PROGRAM MAIN
VAR
	{attribute 'OPC.UA.DA' := '1'}
	{attribute 'OPC.UA.DA.StructuredType' := '1'}
	//Simulate virtual axes
	simulated		:	ARRAY [1..GVL.axisNumMax] OF ST_SimulateStage;
	bSimulate		:	ARRAY [1..GVL.axisNumMax] OF BOOL;	//Do we want to simulate?
	
	//{attribute 'OPC.UA.DA' := '0'}
	drives			:	ARRAY [1..GVL.axisNumMax] OF FB_AxisDrive;	
	
	bDisableMC		:	BOOL; 		//boolean control if true the motion control application specific code is disabled - dumb box
	iState			:	UINT;		//state machine index

	(*
		Outputs that are set in the hmi and wired to power axis limit switches. Currently not configred as part of the programme
		Will be added to ST_AxisControl in future
	*)
	limitEnable1	AT %Q*	: BOOL;
	limitEnable2	AT %Q*	: BOOL;	
	
	i: UINT;		//General indexing value for FOR loops	
	
	//HMI VARIABLES	
	hmiAxisSelect	:	UINT:=1;

END_VAR

AXES();
PROG();
//SIMULATE();

ACTION AXES:
FOR GVL.iAxis:=1 TO GVL.axisNumMax DO
	drives[GVL.iAxis](AxisController:=GVL.axes[GVL.iAxis]);
END_FOR
END_ACTION

(*
	Scans through axes (from low to high) checking "done" status
*)
METHOD CheckCoupled : BOOL
VAR_INPUT
	iLow	:	UINT;		//lowest index to check
	iHigh	:	UINT;		//highest index to check
END_VAR

VAR
	i		:	UINT;
END_VAR
CheckCoupled:=TRUE;
FOR i:=iLow TO iHigh BY 1 DO
	CheckCoupled:= CheckCoupled AND (GVL.axes[i].iAxisState=500);
END_FOR
END_METHOD

(*
	Scans through axes (from low to high) checking "done" status
*)
METHOD CheckDone : BOOL
VAR_INPUT
	iLow	:	UINT;		//lowest index to check
	iHigh	:	UINT;		//highest index to check
END_VAR

VAR
	i		:	UINT;
END_VAR
CheckDone:=TRUE;
FOR i:=iLow TO iHigh BY 1 DO
	CheckDone:= CheckDone AND GVL.axes[i].bDone;
END_FOR
END_METHOD

(*
	Scans through axes (from low to high) checking "done" status
*)
METHOD CheckMoving : BOOL
VAR_INPUT
	iLow	:	UINT;		//lowest index to check
	iHigh	:	UINT;		//highest index to check
END_VAR

VAR
	i		:	UINT;
	statiks: INT;
END_VAR
CheckMoving:=FALSE;
FOR i:=iLow TO iHigh BY 1 DO
	CheckMoving:= CheckMoving OR (GVL.axes[i].Axis.status.Moving);
END_FOR
END_METHOD

(*
	Gear out an axis
*)
METHOD GearOut : BOOL
VAR_INPUT
	i	:	UINT;	//Axis index to gear out
END_VAR
GVL.axes[i].eCommand:=eMcCommand.GearOut;
GVL.axes[i].bExecute:=TRUE;
END_METHOD

(*
	Power up a single axis of index i
*)
METHOD PowerUp : BOOL
VAR_INPUT
	i	:	UINT;
END_VAR
GVL.axes[i].bEnable:=TRUE;
GVL.axes[i].fOverride:=100;
Limits.FwLimit[i]:=TRUE;	//Set high as I have no hardware linked
Limits.BwLimit[i]:=TRUE;	//Set high as I have no hardware linked
END_METHOD

ACTION PROG:
CASE iState OF
	0:	//CHECK AXIS ID's are correct. Gearing limits currently requires the assigned array index of an axis to match the NC ID.
		//May be possible to negate this by changing axes to GVLs so that they can be seen within the drives function - CASE 0 NO LONGER REQ
		iState:=1;
		FOR i:=1 TO GVL.axisNumMax BY 1 DO
			IF GVL.axes[i].Axis.NcToPlc.AxisId <> i THEN
				iState:=999;
			END_IF
		END_FOR
		
	1:	//Gear out all axes to begin
		FOR i:=1 TO 8 BY 1 DO
			GearOut(i:=i);
		END_FOR
		iState:= 2;
	2:	//Wait for gear out
		IF CheckDone(iLow:=1, iHigh:=8) THEN
			iState:=3;
		END_IF
	3:	//Power up axes (and set limits true as no hardware connected)
		limitEnable1 	:=	TRUE;
		limitEnable2	:=	TRUE;
		FOR i:=1 TO 8 BY 1 DO
			PowerUp(i:=i);
		END_FOR
		iState:= 4;
		
	4:	//HOMING ROUTING
		
		iState:=	10;
		
		
	10:	//Start of main state loop. Are the blades coupled in to the virtual axes?
		//SlitPositions(North:=1,South:=2,East:=3,West:=4,VG:=5,VC:=6,HG:=7,HC:=8);
		IF NOT CheckCoupled(iLow:=1, iHigh:=4) THEN
			iState:=11;
		END_IF
		
	11:	//Blades are not coupled. Update the virtual positions
		FOR i:=1 TO 8 BY 1 DO
			GearOut(i:=i);
		END_FOR
	
		iState:=12;
			
		
	12:	//Confirm positions set
		IF CheckDone(iLow:=5,iHigh:=8) THEN
			iState:=12;
		END_IF	
		iState:=13;
	
	13:	//Check Moving
		SlitPositions(North:=1,South:=2,East:=3,West:=4,VG:=5,VC:=6,HG:=7,HC:=8);
		iState:=14;
		

	14: //Blades not moving, time to setup again
		IF CheckDone(iLow:=5,iHigh:=8) THEN
			iState:=15;
		END_IF			

		
	15:	//Check movin
		IF CheckMoving(iLow:=1, iHigh:=4) THEN
			iState:= 13;
		ELSE
			iState:=16;
		END_IF
	

	16:	//Multimaster gearin
		SlitSetup(North:=1,South:=2,East:=3,West:=4,VG:=5,VC:=6,HG:=7,HC:=8);
		iState:=17;	
		
	17:
		IF CheckDone(iLow:=1,iHigh:=8) THEN
			iState:=10;
		END_IF
		
	50:
		
	51:
						
			
	100:	//DO NOTHING

		
	
	999: //ERROR
		//INOP STATE	
END_CASE
END_ACTION

ACTION SIMULATE:
(*
Simulate axes if bool set TRUE
*)
FOR i:=1 TO GVL.axisNumMax BY 1 DO
	IF bSimulate[i] THEN
		simulateStage(position:=GVL.axes[i].Axis.NcToPlc.ActPos, iAxis:=i, simulated:=simulated[i]);
		GVL.axes[i].MCSignalRef.Level:=simulated[i].absSw;
	END_IF
END_FOR
END_ACTION

(*
	Basic virtual axis simulation.
	Will trigger limit switches beyond set points
	Will trigger absolute switch between given set points
*)
METHOD simulateStage : BOOL
VAR_INPUT
	position	:	LREAL;		//Axis current position
	iAxis		:	UINT;		//Axis index
END_VAR
VAR_IN_OUT
	simulated	:	ST_SimulateStage;	//Struct to hold simulation parameters
END_VAR
Limits.FwLimit[iAxis]:= position < simulated.fHighLim;
Limits.BwLimit[iAxis]:= position > simulated.fLowLim;

simulated.absSw:= (position < simulated.fHighAbs) AND (position > simulated.fLowAbs);
END_METHOD

(*
	Calculate gap positions of a slit set given N/S/E/W blades
*)
METHOD SlitPositions : BOOL
VAR_INPUT
	North	:	UINT;	//North blade index
	South	:	UINT;	//South blade index
	East	:	UINT;	//East blade index
	West	:	UINT;	//West blade index
	VG		:	UINT;	//Vertical gap size index
	VC		:	UINT;	//Vertical gap centre index
	HG		:	UINT;	//Horizontal gap size index
	HC		:	UINT;	//Horizontal gap centre index
END_VAR
GVL.axes[VG].eCommand:=eMcCommand.SetPosition;
GVL.axes[VG].fPosition:=GVL.axes[North].Axis.NcToPlc.ActPos-GVL.axes[South].Axis.NcToPlc.ActPos;
GVL.axes[VG].bExecute:=TRUE;

GVL.axes[VC].eCommand:=eMcCommand.SetPosition;
GVL.axes[VC].fPosition:=(GVL.axes[North].Axis.NcToPlc.ActPos+GVL.axes[South].Axis.NcToPlc.ActPos)/2;
GVL.axes[VC].bExecute:=TRUE;

GVL.axes[HG].eCommand:=eMcCommand.SetPosition;
GVL.axes[HG].fPosition:=GVL.axes[East].Axis.NcToPlc.ActPos-GVL.axes[West].Axis.NcToPlc.ActPos;
GVL.axes[HG].bExecute:=TRUE;

GVL.axes[HC].eCommand:=eMcCommand.SetPosition;
GVL.axes[HC].fPosition:=(GVL.axes[East].Axis.NcToPlc.ActPos+GVL.axes[West].Axis.NcToPlc.ActPos)/2;
GVL.axes[HC].bExecute:=TRUE;
END_METHOD

(*
	Gear in blades to gaps for a slit set
*)
METHOD SlitSetup : BOOL
VAR_INPUT
	North	:	UINT;
	South	:	UINT;
	East	:	UINT;
	West	:	UINT;
	VG		:	UINT;
	VC		:	UINT;
	HG		:	UINT;
	HC		:	UINT;
END_VAR
GVL.axes[North].eCommand:= eMcCommand.GearInMultiMaster;
GVL.axes[North].bExecute:=TRUE;
GVL.axes[NORTH].masterAxes[1].i:=VG;
GVL.axes[NORTH].masterAxes[2].i:=VC;
GVL.axes[NORTH].masterAxes[1].ratio:=0.5;
GVL.axes[NORTH].masterAxes[2].ratio:=1;

GVL.axes[South].eCommand:= eMcCommand.GearInMultiMaster;
GVL.axes[South].bExecute:=TRUE;
GVL.axes[South].masterAxes[1].i:=VG;
GVL.axes[South].masterAxes[2].i:=VC;
GVL.axes[South].masterAxes[1].ratio:=-0.5;
GVL.axes[South].masterAxes[2].ratio:=1;

GVL.axes[West].eCommand:= eMcCommand.GearInMultiMaster;
GVL.axes[West].bExecute:=TRUE;
GVL.axes[West].masterAxes[1].i:=HG;
GVL.axes[West].masterAxes[2].i:=HC;
GVL.axes[West].masterAxes[1].ratio:=-0.5;
GVL.axes[West].masterAxes[2].ratio:=1;


GVL.axes[East].eCommand:= eMcCommand.GearInMultiMaster;
GVL.axes[East].bExecute:=TRUE;
GVL.axes[East].masterAxes[1].i:=HG;
GVL.axes[East].masterAxes[2].i:=HC;
GVL.axes[East].masterAxes[1].ratio:=0.5;
GVL.axes[East].masterAxes[2].ratio:=1;
END_METHOD

END_PROGRAM

(* stored: Version 1.1.0.1, ProductVersion 3.1.4022.12
   POU MAIN: Id {0ea98677-ea3a-4346-a22a-d9ad819fe0c1}, SpecialFunc None
   Folder Prog Methods: Id {212990ae-6442-4648-907a-9b74a7c9f90f}
   Folder Simulate Methods: Id {9564da1a-4827-4610-81ab-1f383f22c9b4}
   Action AXES: Id {64e9147a-f428-4655-bd0f-63c28bb82a85}
   Method CheckCoupled: Id {3f7a8e9f-d86f-408a-ae71-3cd4846c79cb}
   Method CheckDone: Id {f8255e59-df7b-4af9-ada6-58c21bf850b3}
   Method CheckMoving: Id {a1b13969-2a4d-43d0-85b1-1b3debcd7e83}
   Method GearOut: Id {c096e6fc-812d-4259-8c64-f354d37770ae}
   Method PowerUp: Id {efa4560c-311a-41aa-bbe0-0aa4eef16646}
   Action PROG: Id {a83d747a-28b8-44b3-812d-dbc6c7a4a77b}
   Action SIMULATE: Id {3ab21edf-3a61-475f-a4eb-e4bcda8bf9cd}
   Method simulateStage: Id {deb827a7-c982-4c31-9561-f2bd7c832d23}
   Method SlitPositions: Id {acef6351-9f47-442e-b66f-59c55dd95878}
   Method SlitSetup: Id {9c346981-cc2d-43a8-b095-88fcece736bc} *)
